(* PLC project conveyors, Dassault Systèmes ControlBuild 2024x Refresh1 *)
(* stored: creationDateTime 2024-04-15T14:49:54-01:00 *)

PROGRAM flask_motion_app.conveyors
  VAR_INPUT
    forwardUp : BOOL := false;
    backwardUp : BOOL := false;
  END_VAR
  VAR_INPUT
    forwardDw : BOOL := false;
    backwardDw : BOOL := false;
  END_VAR
  VAR_INPUT
    ejectBadProd : BOOL := false;
  END_VAR
  VAR_OUTPUT
    presConvUp : BOOL := false;
    presConvDw : BOOL := false;
    idRead : INT := 0;
    mesuredWeight : INT := 0;
  END_VAR
  VAR_OUTPUT
    bpStart : BOOL := false;
    bpAuto : BOOL := false;
    bpManu : BOOL := false;
    bpEmergencyStop : BOOL := false;
    bpStop : BOOL := false;
  END_VAR

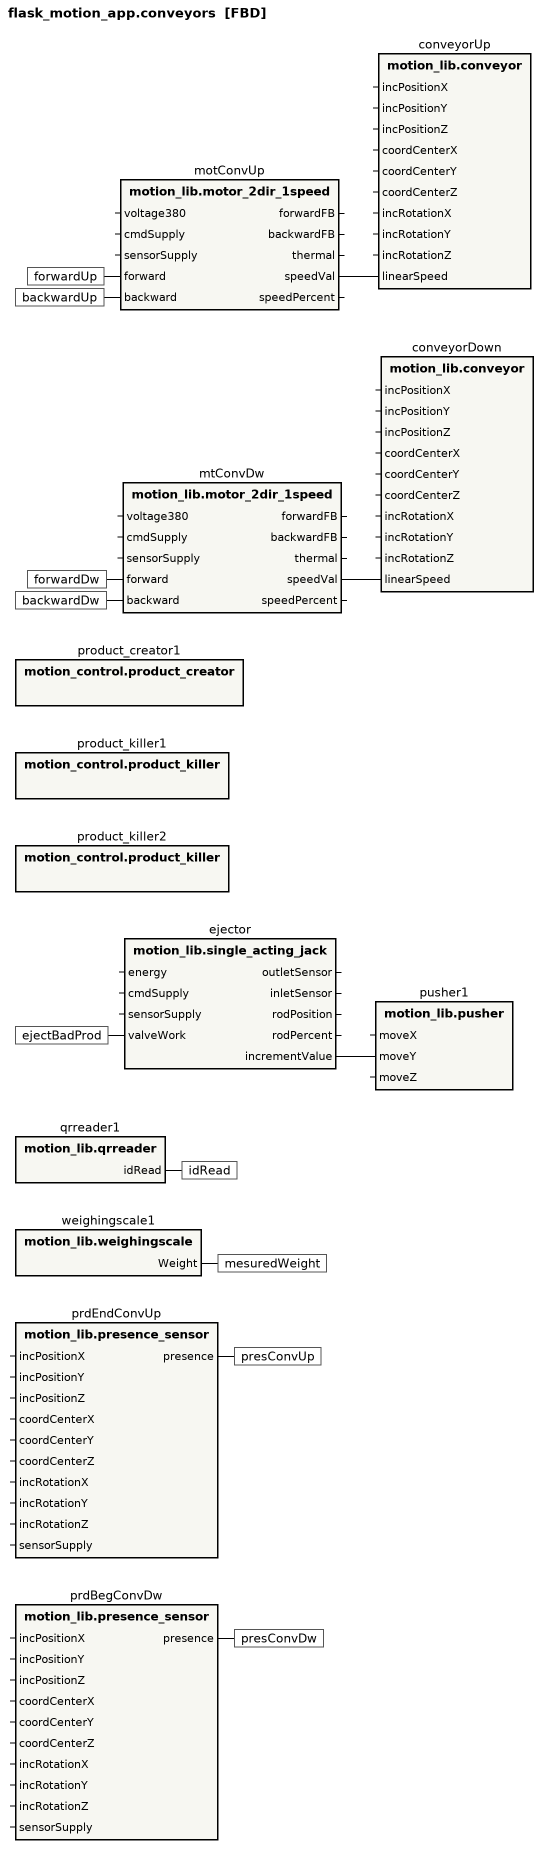
(* FBD diagram, written out as Structured Text *)
prdEndConvUp();
presConvUp := prdEndConvUp.presence;
prdBegConvDw();
presConvDw := prdBegConvDw.presence;
qrreader1();
idRead := qrreader1.idRead;
weighingscale1();
mesuredWeight := weighingscale1.Weight;
motConvUp(forward := forwardUp, backward := backwardUp);
conveyorUp(linearSpeed := motConvUp.speedVal);
mtConvDw(forward := forwardDw, backward := backwardDw);
conveyorDown(linearSpeed := mtConvDw.speedVal);
product_creator1();
product_killer1();
product_killer2();
ejector(valveWork := ejectBadProd);
pusher1(moveY := ejector.incrementValue);
END_PROGRAM
